// Writes an sfixed32 value, without a tag, to the stream.
FUNCTION F_WriteSFixed32 : HRESULT
VAR_IN_OUT      
    stCtx : ST_WriteContext;
END_VAR
VAR_INPUT
    nValue : DINT;
END_VAR
VAR
END_VAR

F_WriteSFixed32 := F_WriteRawLittleEndian32(stCtx, TO_UDINT(nValue));

END_FUNCTION

(* stored: Version 1.1.0.1
   POU F_WriteSFixed32: Id {1954aae2-e95c-4dac-8af1-a579da471d1b}, SpecialFunc None *)
